# EPICS substitutions: db/Beckhoff_KL/ecmcBK1150.substitutions
file "ecmcEcSlave.template"
{
  pattern {}
          {}
}

file "ecmcBK1X50.template"
{
  pattern {}
          {}
}
